PROGRAM MAIN
VAR
	
	Drill	:	DataDrill;
	Drill2	:	DataDrill;

	nState: INT;
	ftrigA: F_TRIG;
	
	rtrigA: R_TRIG;
	
	ftrigB: F_TRIG;
	ftrigUON: F_TRIG;
	
	fDrillY: REAL;
	C: BOOL;
END_VAR


C	:=	NOT(Drill.IN.bSwitchC);

ACT_MatkapUygulamasi();
ACT_Visu();

ACTION ACT_MatkapUygulamasi:

rtrigA(CLK:= Drill.IN.bSwitchA , Q=> );
ftrigA(CLK:= Drill.IN.bSwitchA , Q=> );


ftrigB(CLK:= Drill.IN.bSwitchB , Q=> );
ftrigUON(CLK:= Drill.IN.bUpSwitch , Q=> );



CASE nState OF
	

	0:
	
		Drill.OUT.bDown	:=	FALSE;
		Drill.OUT.bUp	:=	FALSE;
	
		IF Drill.IN.bStart AND 
		NOT Drill.IN.bUpSwitch AND
		 Drill.IN.bSwitchC	THEN
		 
			nState := 10;
		
		END_IF
	
		
	10:
		
		Drill.OUT.bDown	:=	TRUE;
		
		IF rtrigA.Q AND Drill.IN.bSwitchC THEN
			
			nState := 20;
			
		ELSIF NOT Drill.IN.bSwitchC THEN
			
			nState := 999;
			
		END_IF
	
		
	20:	
	
		Drill.OUT.bDrill	:=	TRUE;
		
		
		IF ftrigB.Q AND Drill.IN.bSwitchC THEN
			
			nState := 30;
			
		ELSIF NOT Drill.IN.bSwitchC THEN
			
			nState := 999;
			
		END_IF	
	
	30:
	
		Drill.OUT.bDown	:=	FALSE;
		Drill.OUT.bUp	:=	TRUE;
	
		IF ftrigA.Q  AND Drill.IN.bSwitchC THEN 

			nState := 40;
			
		ELSIF NOT Drill.IN.bSwitchC THEN
		
			nState := 999;
			
		END_IF
		
	40:
	
		Drill.OUT.bDrill	:=	FALSE;

		IF ftrigUON.Q THEN
			
		Drill.OUT.bDown	:=	FALSE;
		Drill.OUT.bUp	:=	FALSE;
		
			nState := 0;
			
		END_IF
	

END_CASE



	IF NOT Drill.IN.bStart	THEN  
			 
		nState := 0;
		Drill.OUT.bDown	:=	FALSE;
		Drill.OUT.bUp	:=	FALSE;		
		Drill.OUT.bDrill	:=	FALSE;
	
	END_IF
END_ACTION

ACTION ACT_Visu:


//50-225

IF Drill.OUT.bDown AND NOT Drill.OUT.bUp THEN
	
	fDrillY	:=	fDrillY + 0.5;
	
	IF fDrillY	>=	100 AND NOT Drill.OUT.bDrill THEN
		fDrillY	:=	100;
	
	
	ELSIF Drill.OUT.bDrill THEN
	
		fDrillY	:=	fDrillY + 0.3;
		
	IF fDrillY	>=	200	THEN
		
		fDrillY	:=	200;
		
	END_IF
	
	END_IF
	

	
ELSIF Drill.OUT.bUp AND NOT Drill.OUT.bDown AND Drill.OUT.bDrill THEN
	
	fDrillY	:=	fDrillY	-	0.3;
	
	IF fDrillY	<=	50	THEN
		fDrillY	:=	50;
	END_IF	

ELSIF Drill.OUT.bUp AND NOT Drill.OUT.bDown AND NOT Drill.OUT.bDrill THEN
	
	fDrillY	:=	fDrillY	-	0.5;
	
	IF fDrillY	<=	20	THEN
		
		fDrillY	:=	20;
		
	END_IF	
	
	
END_IF
END_ACTION

END_PROGRAM

(* stored: Version 1.1.0.1, ProductVersion 3.1.4024.4
   POU MAIN: Id {536253be-ada7-4d6d-a05b-554eeb256f50}, SpecialFunc None
   Action ACT_MatkapUygulamasi: Id {c679b45d-7911-4797-9d2e-c2916cb9a363}
   Action ACT_Visu: Id {505970fd-13c2-471c-9c6b-051a6fa818f2} *)
